FUNCTION_BLOCK FB_SafetyManager
VAR

END_VAR

END_FUNCTION_BLOCK

(* stored: Version 1.1.0.1, ProductVersion 3.1.4026.18
   POU FB_SafetyManager: Id {1c642676-d698-4f2b-b05b-dc3832527b44}, SpecialFunc None *)
